FUNCTION_BLOCK "GetSomeBullshit"
{ S7_Optimized_Access := 'TRUE' }
VERSION : 0.1
   VAR
      Auch { S7_SetPoint := 'False'} : "Anwenderdatentyp_1";
      Und : "Anwenderdatentyp_1";
   END_VAR


BEGIN
	(* 1st edit *)
	(* 2nd edit *)
	(* 3rd edit *)
	(* 4th edit *)
END_FUNCTION_BLOCK

